FUNCTION_BLOCK L2_Alimentador_SFC EXTENDS L1_ControllerBase_SFC

VAR_INPUT 					// Sensores y comandos
	k1	: BOOL; 			// Sensor de empujador tapa delante
	Alimentar :BOOL;
END_VAR

VAR_OUTPUT					// Actuadores
	Leyendo: BOOL;	
	K_1: BOOL; 				// Actuador de empujador tapa avanza	 
	FM : BOOL; 
END_VAR

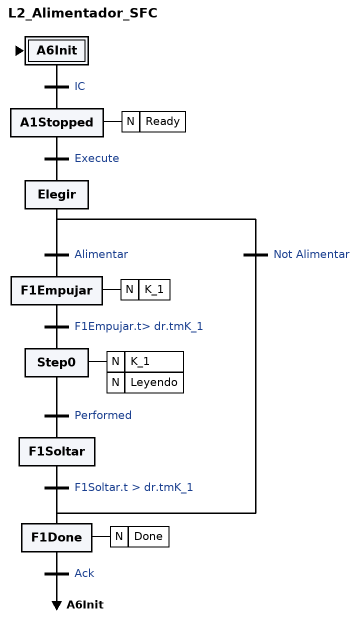
INITIAL_STEP A6Init:
END_STEP
TRANSITION FROM A6Init TO A1Stopped
    := IC;
END_TRANSITION
STEP A1Stopped:
    Ready(N);
END_STEP
TRANSITION FROM A1Stopped TO Elegir
    := Execute;
END_TRANSITION
STEP Elegir:
END_STEP
TRANSITION FROM Elegir TO F1Empujar
    := Alimentar;
END_TRANSITION
STEP F1Empujar:
    K_1(N);
END_STEP
TRANSITION FROM F1Empujar TO Step0
    := F1Empujar.t> dr.tmK_1;
END_TRANSITION
STEP Step0:
    K_1(N);
    Leyendo(N);
END_STEP
TRANSITION FROM Step0 TO F1Soltar
    := Performed;
END_TRANSITION
STEP F1Soltar:
END_STEP
TRANSITION FROM F1Soltar TO F1Done
    := F1Soltar.t > dr.tmK_1;
END_TRANSITION
TRANSITION FROM Elegir TO F1Done
    := Not Alimentar;
END_TRANSITION
STEP F1Done:
    Done(N);
END_STEP
TRANSITION FROM F1Done TO A6Init
    := Ack;
END_TRANSITION

END_FUNCTION_BLOCK

(* stored: Version 1.1.0.1, ProductVersion 3.1.4024.6
   POU L2_Alimentador_SFC: Id {25ad7b61-92b1-41db-8b65-16e3fd2054f3}, SpecialFunc None *)
